(* IEC 61131-3 sources: repolevel_ST_code_completion/output/0121完整版本/repoeval_Command1/readful_result, 11 files *)

(* ---- FB_AirConComfortCommand.st ---- *)
FUNCTION_BLOCK PUBLIC FB_AirConComfortCommand IMPLEMENTS I_Command
VAR
	refAirConditioning : REFERENCE TO FB_AirConditioning;
END_VAR

METHOD Execute : BOOL
VAR
	isValid : BOOL;
END_VAR

isValid := (refAirConditioning <> 0);

IF isValid THEN
refAirConditioning^.Activate();
refAirConditioning^.SetTemperature(20.0);
Execute := TRUE;
ELSE
Execute := FALSE;
END_IF
END_FUNCTION_BLOCK

(* ---- FB_AirConStandbyCommand.st ---- *)
FUNCTION_BLOCK FB_AirConStandbyCommand IMPLEMENTS I_Command
VAR
  refAirConditioning : REFERENCE TO FB_AirConditioning;
END_VAR

IF __ISVALIDREF(refAirConditioning) THEN
  refAirConditioning.bActive := FALSE;
END_IF
END_FB

(* ---- FB_CDPlayer.st ---- *)
FUNCTION_BLOCK PUBLIC FB_CDPlayer
VAR_OUTPUT
bPlayerActive		: BOOL;
byVolume			: BYTE;
byTrack				: UINT;
END_VAR
VAR
bInitialized        : BOOL := FALSE;
END_VAR

IF NOT bInitialized THEN
bPlayerActive := FALSE;
byVolume := 50; // Default volume level
byTrack := 1;   // Default track number
bInitialized := TRUE;
END_IF

IF bPlayerActive THEN
// Player is active, maintain current state
// No action needed here; bPlayerActive is already TRUE
ELSE
// Player is inactive, reset outputs
byVolume := 0;
byTrack := 0;
END_IF;
END_FUNCTION_BLOCK

(* ---- FB_Lamp.st ---- *)
FUNCTION_BLOCK PUBLIC FB_Lamp
VAR_OUTPUT
	byLevel			: BYTE;
END_VAR
VAR
    byCurrentLevel : BYTE := 0;
END_VAR

IF byCurrentLevel <> byLevel THEN
    byCurrentLevel := byLevel;
END_IF
END_FUNCTION_BLOCK

(* ---- FB_LampSetLevelCommand.st ---- *)
FUNCTION_BLOCK PUBLIC FB_LampSetLevelCommand IMPLEMENTS I_Command
VAR
	refLamp		: REFERENCE TO FB_Lamp;
	byNewLevel	: BYTE;
END_VAR

METHOD Execute : BOOL
VAR
	isSuccessful : BOOL;
END_VAR

IF __ISVALIDREF(refLamp) THEN
 // Directly assign the result of SetLevel to Execute
 IF refLamp.SetLevel(byNewLevel) THEN
  Execute := TRUE;
 ELSE
  Execute := FALSE;
 END_IF;
ELSE
 Execute := FALSE;
END_IF
END_FUNCTION_BLOCK

(* ---- FB_MusicPlayCommand.st ---- *)
FUNCTION_BLOCK PUBLIC FB_MusicPlayCommand IMPLEMENTS I_Command
VAR
    refCDPlayer : REFERENCE TO FB_CDPlayer;
END_VAR

METHOD Execute
VAR
END_VAR

IF (__ISVALIDREF(refCDPlayer)) THEN
  refCDPlayer.SetVolume(40);
  refCDPlayer.SetTrack(1);
  refCDPlayer.Start();
END_IF
END_FUNCTION_BLOCK

(* ---- FB_MusicStopCommand.st ---- *)
FUNCTION_BLOCK PUBLIC FB_MusicStopCommand IMPLEMENTS I_Command
VAR
	refCDPlayer : REFERENCE TO FB_CDPlayer;
END_VAR

METHOD Execute
// Removed redundant re-declaration of refCDPlayer to fix the shadowing error.

IF (__ISVALIDREF(THIS^.refCDPlayer)) THEN
  THIS^.refCDPlayer.Stop();
END_IF
END_FUNCTION_BLOCK

(* ---- FB_Socket.st ---- *)
FUNCTION_BLOCK PUBLIC FB_Socket
VAR_OUTPUT
 bActive		: BOOL;
END_VAR
VAR
 bInitialized : BOOL := FALSE;
END_VAR

METHOD PUBLIC Main : VOID
IF NOT bInitialized THEN
 bActive := FALSE;
 bInitialized := TRUE;
END_IF
END_METHOD
END_FUNCTION_BLOCK

(* ---- FB_SocketOffCommand.st ---- *)
FUNCTION_BLOCK PUBLIC FB_SocketOffCommand IMPLEMENTS I_Command
VAR
  refSocket : REFERENCE TO FB_Socket;
END_VAR

IF __ISVALIDREF(refSocket) THEN
  refSocket.Off();
END_IF
END_FUNCTION

(* ---- FB_SocketOnCommand.st ---- *)
FUNCTION_BLOCK PUBLIC FB_SocketOnCommand IMPLEMENTS I_Command
VAR
refSocket : REFERENCE TO FB_Socket;
END_VAR

METHOD Execute
VAR
END_VAR
IF (__ISVALIDREF(refSocket)) THEN
refSocket^.bActive := TRUE;
END_IF
END_FUNCTION_BLOCK

(* ---- FB_SwitchPanel.st ---- *)
FUNCTION_BLOCK PUBLIC FB_SwitchPanel
VAR_INPUT
	arrSwitch		: ARRAY[1..8] OF BOOL;
END_VAR
VAR
	aiCommand		: ARRAY[1..8] OF I_Command;
	arrRtrig		: ARRAY[1..8] OF R_TRIG;
	nIndex			: INT;
END_VAR

FOR nIndex := 1 TO 8 DO
  arrRtrig[nIndex](CLK := arrSwitch[nIndex]);
  IF arrRtrig[nIndex].Q THEN
    aiCommand[nIndex].Execute(); // Execute method of the initialized function block
  END_IF
END_FOR
END_FUNCTION_BLOCK
